TYPE E_RevSeq : (
		Stopped,
		Move1,
		Wait1,
		Idle1,
		Move2,
		Wait2,
		Idle2,
		Error
	) INT;
END_TYPE

(* stored: Version 1.1.0.1, ProductVersion 3.1.4024.13
   DUT E_RevSeq: Id {e5213198-d12f-4857-bb58-bafe9a6dda27} *)
